Omron Sysmac Studio project NX1P2_MQTT_Demo_3 (Sysmac Studio 1.45.1.64010, StandardProject)

# Controller new_Controller_0: NX1P2-9024DT version 1.40
Task PrimaryTask (priority 4, period or condition 2000): Program0
Library MQTT 0.44.98f 0.44.98 (contents left out)
Library JSON 0.0.55 (contents left out)

VAR_GLOBAL
    cam1 : ARRAY[0..1000] OF _sMC_CAM_REF := None;
    input : int;  (* published *)
END_VAR

PROGRAM Program0
VAR
    Move_1 : MC_MoveRelative;
    Move_2 : MC_MoveRelative;
    ulTimeInStop : ULINT;
    Start : BOOL;
    Cam_1 : MC_CamIn;
    RandomValue : LREAL;
    RandomFailure : Rand;
    RandomSpeed : LREAL;
    RandomStop : LREAL;
    OtherStop : BOOL;
    ErrorStop : BOOL;
    Velocity : LREAL;
    MasterReference : MC_MoveVelocity;
    MasterStop : MC_Stop;
    StopStatus : BOOL;
    TimeInStop : TIME;
    Timer_Stop : TON;
    TimeStopCounter : AccumulationTimer;
    TimeALL : AccumulationTimer;
    accTimeInStop : TIME;
    accTime : TIME;
    Reset : BOOL;
    Availability : LREAL;
    M : BOOL;
    TotalProduction : UDINT;
    TotalProductionNG : UDINT;
    Quality : LREAL;
    curProductionHour : LREAL;
    Performance : LREAL;
    OEE : LREAL;
    JSON_OEE : JSON\JSONBuffer;
    JSON_MachineData : JSON\JSONBuffer;
    JSON_Events : JSON\JSONBuffer;
    TimeStamp : DATE_AND_TIME;
    MQTT_Client : MQTT\MQTTClient;
    UserLogin : MQTT\Login;
    DataBuffer : MQTT\ClientBuffer;
    Host : STRING[256];
    ServerPort : UINT;
    machineOEE : STRING[64];
    BrokerConnect : BOOL;
    Publish_OEE : MQTT\MQTTPublish;
    Publish_MachineData : MQTT\MQTTPublish;
    Publish_Events : MQTT\MQTTPublish;
    test : BOOL;
    openSkt : SktTCPConnect;
    ElapsedTime : LREAL;
    SendEvent : BOOL;
    se : BOOL;
    x : BOOL;
    Subscribe : BOOL;
    MQTTSubscribe : MQTT\MQTTSubscribe;
    Subscribe_Temperature : MQTT\MQTTSubscribe;
    Subscribe_Humidity : MQTT\MQTTSubscribe;
    strTemperature : STRING[256];
    strHumidity : STRING[256];
    txtJSON_OEE : STRING[1856];
    txtJSON_MachineData : STRING[1856];
    txtJSON_Events : string[1856];
    bConInit : BOOL;
    uiConnection : UINT;
    bWait : BOOL;
    bReconnect : BOOL;
    uiConnectionAttempt : UINT;
    T_Reconnection : TON;
    T_Wait : TON;
    Timer_Start : TON;
    ErrorIDex : DWORD;
    LWC : MQTT\WillCnfg;
    lwt : MQTT\WillCnfg;
    WelcomeMessage : MQTT\MQTTPublish;
    Welcome : STRING[1986];
    MQTT_ping : MQTT\MQTTPing;
    ServerAlive : BOOL;
    ResponseTime : UINT;
    Busy : BOOL;
END_VAR
VAR_EXTERNAL
    cam1 : ARRAY[0..1000] OF _sMC_CAM_REF;
END_VAR
VAR_EXTERNAL CONSTANT
    _EIP_EtnOnlineSta : BOOL;
END_VAR
VAR
    _e1 : R_TRIG;
    _e2 : R_TRIG;
    _e3 : F_TRIG;
    _e4 : R_TRIG;
    _e5 : F_TRIG;
    _e6 : R_TRIG;
    _e7 : R_TRIG;
END_VAR

(* Section M_OEE: ladder, written here as Structured Text *)

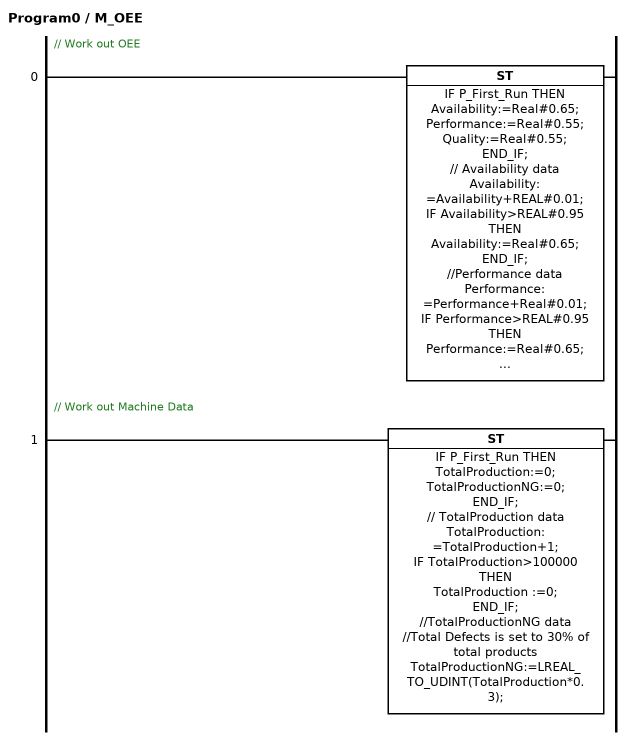
(* Rung 0: // Work out OEE *)
IF P_First_Run THEN
Availability:=Real#0.65;
Performance:=Real#0.55;
Quality:=Real#0.55;
END_IF;

// Availability data
Availability:=Availability+REAL#0.01;

IF Availability>REAL#0.95 THEN
	Availability:=Real#0.65;
END_IF;

//Performance data
Performance:=Performance+Real#0.01;

IF Performance>REAL#0.95 THEN
	Performance:=Real#0.65;
END_IF;

//Quality data
Quality:=Quality+Real#0.01;

IF Quality>REAL#0.90 THEN
	Quality:=Real#0.55;
END_IF;
	
OEE:=Availability*Performance*Quality; 
(* Rung 1: // Work out Machine Data *)
IF P_First_Run THEN
TotalProduction:=0;
TotalProductionNG:=0;
END_IF;

// TotalProduction data
TotalProduction:=TotalProduction+1;

IF TotalProduction>100000 THEN
	TotalProduction :=0;
END_IF;

//TotalProductionNG data
//Total Defects is set to 30% of total products
TotalProductionNG:=LREAL_TO_UDINT(TotalProduction*0.3);

(* Section Data_Collection: ladder, written here as Structured Text *)

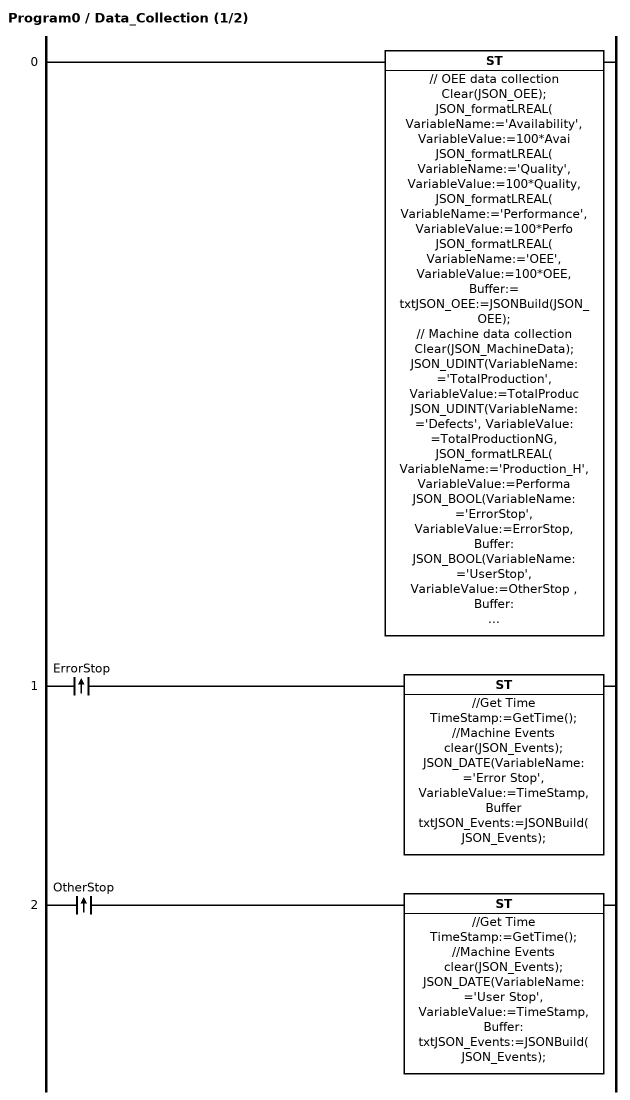
(* Rung 0 *)
// OEE data collection
Clear(JSON_OEE);
JSON_formatLREAL(VariableName:='Availability', VariableValue:=100*Availability, Buffer:=JSON_OEE, MinLen:=3, DecPlace:=1);
JSON_formatLREAL(VariableName:='Quality', VariableValue:=100*Quality, Buffer:=JSON_OEE, MinLen:=3, DecPlace:=1);
JSON_formatLREAL(VariableName:='Performance', VariableValue:=100*Performance, Buffer:=JSON_OEE, MinLen:=3, DecPlace:=1);
JSON_formatLREAL(VariableName:='OEE', VariableValue:=100*OEE, Buffer:=JSON_OEE, MinLen:=3, DecPlace:=1);
txtJSON_OEE:=JSONBuild(JSON_OEE);

// Machine data collection
Clear(JSON_MachineData);
JSON_UDINT(VariableName:='TotalProduction', VariableValue:=TotalProduction, Buffer:=JSON_MachineData);
JSON_UDINT(VariableName:='Defects', VariableValue:=TotalProductionNG, Buffer:=JSON_MachineData);
JSON_formatLREAL(VariableName:='Production_H', VariableValue:=Performance*3600, Buffer:=JSON_MachineData);
JSON_BOOL(VariableName:='ErrorStop', VariableValue:=ErrorStop, Buffer:=JSON_MachineData);
JSON_BOOL(VariableName:='UserStop', VariableValue:=OtherStop , Buffer:=JSON_MachineData);
JSON_BOOL(VariableName:='InOperation', VariableValue:=NOT(StopStatus) , Buffer:=JSON_MachineData);
txtJSON_MachineData:=JSONBuild(JSON_MachineData);
(* Rung 1 *)
_e1(CLK := ErrorStop);
IF _e1.Q THEN
    //Get Time
    TimeStamp:=GetTime();
    
    //Machine Events
    clear(JSON_Events);
    JSON_DATE(VariableName:='Error Stop', VariableValue:=TimeStamp, Buffer:=JSON_Events);
    txtJSON_Events:=JSONBuild(JSON_Events);
END_IF;
(* Rung 2 *)
_e2(CLK := OtherStop);
IF _e2.Q THEN
    //Get Time
    TimeStamp:=GetTime();
    
    //Machine Events
    clear(JSON_Events);
    JSON_DATE(VariableName:='User Stop', VariableValue:=TimeStamp, Buffer:=JSON_Events);
    txtJSON_Events:=JSONBuild(JSON_Events);
END_IF;

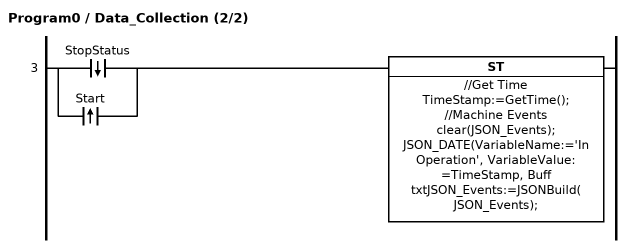
(* Rung 3 *)
_e3(CLK := StopStatus);
_e4(CLK := Start);
IF _e3.Q OR _e4.Q THEN
    //Get Time
    TimeStamp:=GetTime();
    
    //Machine Events
    clear(JSON_Events);
    JSON_DATE(VariableName:='In Operation', VariableValue:=TimeStamp, Buffer:=JSON_Events);
    txtJSON_Events:=JSONBuild(JSON_Events);
END_IF;

(* Section MQTT_client: ladder, written here as Structured Text *)

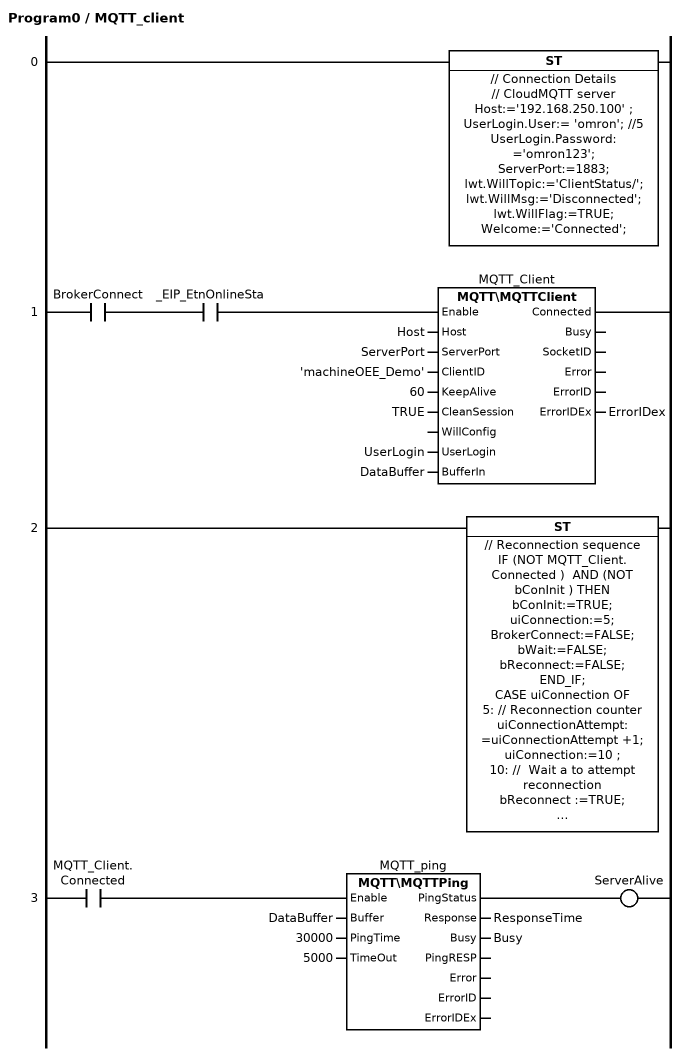
(* Rung 0 *)
// Connection Details
// CloudMQTT server 
Host:='192.168.250.100' ;
UserLogin.User:= 'omron'; //5
UserLogin.Password:='omron123';
ServerPort:=1883;

lwt.WillTopic:='ClientStatus/';
lwt.WillMsg:='Disconnected';
lwt.WillFlag:=TRUE;

Welcome:='Connected';
(* Rung 1 *)
MQTT_Client(Enable := BrokerConnect AND _EIP_EtnOnlineSta, Host := Host, ServerPort := ServerPort, ClientID := 'machineOEE_Demo', KeepAlive := 60, CleanSession := TRUE, UserLogin := UserLogin, BufferIn := DataBuffer, ErrorIDEx => ErrorIDex);
(* Rung 2 *)
// Reconnection sequence
IF (NOT MQTT_Client.Connected )  AND (NOT bConInit ) THEN
	bConInit:=TRUE;
	uiConnection:=5;
	BrokerConnect:=FALSE;
	bWait:=FALSE;
	bReconnect:=FALSE;
END_IF;

CASE uiConnection OF
	
	5: // Reconnection counter	
		uiConnectionAttempt:=uiConnectionAttempt +1;
		uiConnection:=10 ;
		
	10: //  Wait a to attempt reconnection
			
			bReconnect :=TRUE;
			IF T_Reconnection.Q THEN
				BrokerConnect:=TRUE;
				bReconnect :=FALSE;
				uiConnection:=20 ;
			END_IF;
			
	20:// Wait a few to see if it connects again
	
				bWait  :=TRUE;
				IF T_Wait .Q AND MQTT_Client.Connected THEN
					// Connection Resumed
					bWait:=FALSE;
					bReconnect:=FALSE;
					bConInit:=false;
					uiConnection:=0;
				ELSIF T_Wait .Q AND NOT MQTT_Client.Connected THEN
					// Connection Refused , new attempt
					uiConnection:=5 ;
					bWait:=FALSE;
					bReconnect:=FALSE;
					BrokerConnect:=FALSE;
				END_IF;
			
	
END_CASE;


// Timers

T_Reconnection(In:=bReconnect, PT:=t#5s );
T_Wait(In:=bWait, PT:=t#10s);


	
	
	
(* Rung 3 *)
MQTT_ping(Enable := MQTT_Client.Connected, Buffer := DataBuffer, PingTime := 30000, TimeOut := 5000, Response => ResponseTime, Busy => Busy);
ServerAlive := MQTT_ping.PingStatus;

(* Section MQTT_Pub: ladder, written here as Structured Text *)

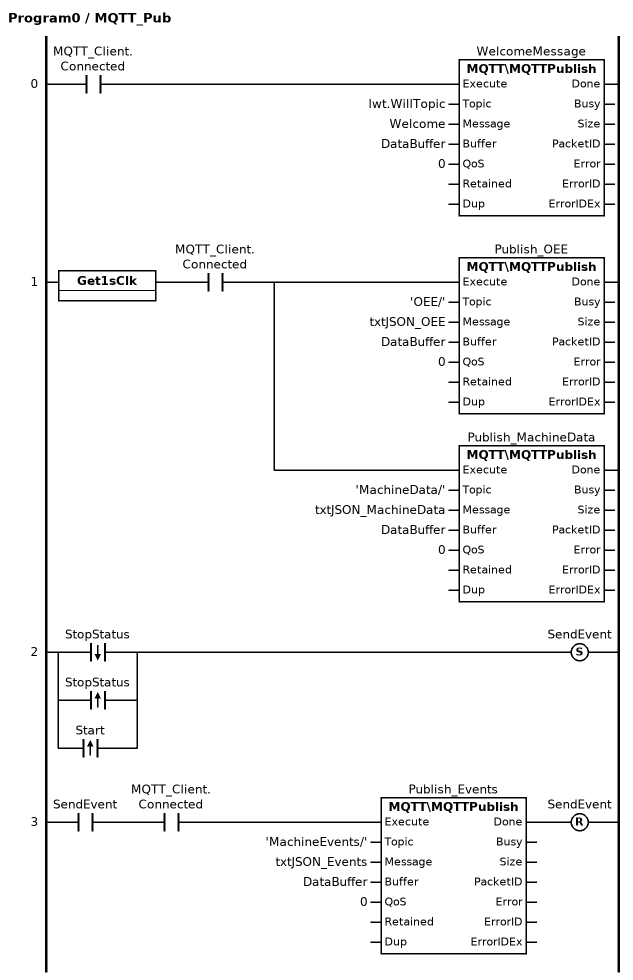
(* Rung 0 *)
WelcomeMessage(Execute := MQTT_Client.Connected, Topic := lwt.WillTopic, Message := Welcome, Buffer := DataBuffer, QoS := 0);
(* Rung 1 *)
Publish_OEE(Execute := Get1sClk() AND MQTT_Client.Connected, Topic := 'OEE/', Message := txtJSON_OEE, Buffer := DataBuffer, QoS := 0);
Publish_MachineData(Execute := Get1sClk() AND MQTT_Client.Connected, Topic := 'MachineData/', Message := txtJSON_MachineData, Buffer := DataBuffer, QoS := 0);
(* Rung 2 *)
_e5(CLK := StopStatus);
_e6(CLK := StopStatus);
_e7(CLK := Start);
IF _e5.Q OR _e6.Q OR _e7.Q THEN SendEvent := TRUE; END_IF;
(* Rung 3 *)
Publish_Events(Execute := SendEvent AND MQTT_Client.Connected, Topic := 'MachineEvents/', Message := txtJSON_Events, Buffer := DataBuffer, QoS := 0);
IF Publish_Events.Done THEN SendEvent := FALSE; END_IF;

(* Section MQTT_Sub: ladder, written here as Structured Text *)

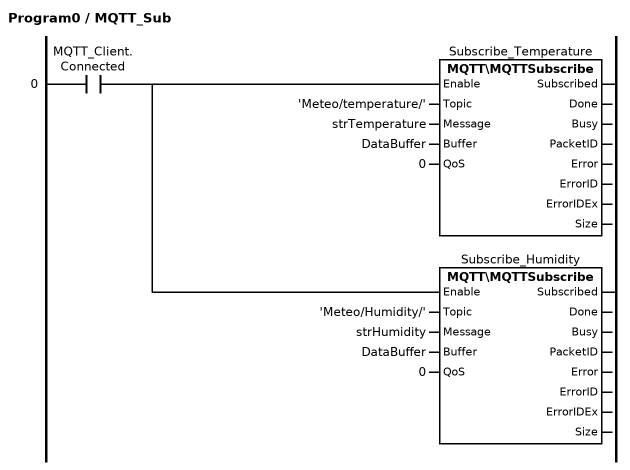
(* Rung 0 *)
Subscribe_Temperature(Enable := MQTT_Client.Connected, Topic := 'Meteo/temperature/', Message := strTemperature, Buffer := DataBuffer, QoS := 0);
Subscribe_Humidity(Enable := MQTT_Client.Connected, Topic := 'Meteo/Humidity/', Message := strHumidity, Buffer := DataBuffer, QoS := 0);
END_PROGRAM